FUNCTION_BLOCK FB_Kierownica
VAR_INPUT
	
			b_czujnik_wejsciowy 	:BOOL;
			b_czujnik_K1 			:BOOL;
			b_czujnik_K2 			:BOOL;
			b_czujnik_K3 			:BOOL;
			b_czujnik_K4 			:BOOL;
			b_czujnik_K5 			:BOOL;
			b_Kon2 					:BOOL;
			b_Kon1 					:BOOL;
			Zasilanie				:BOOL;
			b_Start					:BOOL;
			b_Start1				:BOOL;
			b_Stop					:BOOL;
			bS_Ready				:BOOL;
			bS_Run					:BOOL;
			bS_Done					:BOOL;
			LR_Pozycja_Zadana				:ARRAY[1..5] OF LREAL;
			b_Pobral 				:BOOL;
			int_Licznik_zadana      :INT;
			int_Kieszen_zadana 		:INT;
			automat					:BOOL;
END_VAR
VAR_OUTPUT
	
			LR_EPozycja				:LREAL;
			LR_Predkosc				:LREAL;
			bS_Enable				:BOOL;
			bS_Exe					:BOOL;
			b_Odbierz				:BOOL;
			b_Hamulec1 				:BOOL;
			b_Hamulec2 				:BOOL;
			Kier_CCW				:BOOL;
			Kier_CW					:BOOL;
END_VAR
VAR
	
			int_Kieszen				:INT :=1;
			int_Licznik				:INT; //liczenie ktora butelka w kasecie
			int_LicznikCheck		:ARRAY[1..5] OF INT; //liczenie ktora butelka w kasecie
			czas					:ARRAY[0..100] OF TON;
			Seq						:INT;
			Seq1						:INT;
			zaladowal				:BOOL;
	i: INT;
END_VAR

LR_Pozycja_Zadana[1]:=-115;	
LR_Pozycja_Zadana[2]:=-53;
LR_Pozycja_Zadana[3]:=7;
LR_Pozycja_Zadana[4]:=63;
LR_Pozycja_Zadana[5]:=122;


CASE seq OF
	

	0:
		//int_Kieszen:=1;
		
	IF (b_Start=TRUE OR b_Start1=TRUE)  AND bS_Ready=TRUE AND Zasilanie=TRUE  THEN
		b_Hamulec1:=TRUE;
		b_Hamulec2:=TRUE;
		
		IF bS_Ready=FALSE THEN 
			
			bS_Enable:=TRUE;
		END_IF
		
		
		IF bS_Ready=TRUE THEN
			seq:=5;
		END_IF
	
	
	END_IF
	
	
	5:
	
	
	
	LR_EPozycja:=LR_Pozycja_Zadana[int_Kieszen];
	LR_Predkosc:=350;
	b_Start:=FALSE;

	IF  b_Kon1=TRUE AND b_Kon2=TRUE THEN
	bS_Exe:=TRUE;
	END_IF
	
	IF bS_Run=TRUE THEN
	seq:=10;

	END_IF
	
	10:
	IF bS_Done=TRUE THEN
	bS_Exe:=FALSE;
	
	IF b_Odbierz=FALSE	THEN 
		b_Hamulec1:=FALSE;
		b_Hamulec2:=FALSE;
		
		END_IF
	seq:=0;
	
	END_IF
	


	
	
END_CASE
CASE seq1 OF
0:

			b_Start:=TRUE;
			seq1:=3;

3:
			//IF Czas[0].Q=FALSE THEN
				
			seq1:=5;
			
			//END_IF
			//int_Licznik	:=0;//zerowanie kieszeni 
			
			
5:

			IF Czas[0].Q=TRUE THEN
				
			seq1:=10;
			
			END_IF
			
10://inkremetnowanie licznika przejchala butelka 
			
			int_Licznik:=int_Licznik+1; 
			seq1:=15;
15:	
			IF int_Licznik=int_Licznik_zadana AND int_Kieszen<int_Kieszen_zadana+1 THEN
			int_Kieszen:=int_Kieszen+1;
			int_Licznik:=0;
			
			seq1:=25;	
			
			
			END_IF
		
	
			IF int_Kieszen=int_Kieszen_zadana+1 THEN
					
			GVL_GLOBAL.reset_licznik:=TRUE; ///moje
			
				b_Odbierz:=TRUE;
				int_Kieszen:=1;
				seq1:=25;	
			END_IF

			
			IF Czas[6].Q=TRUE THEN
			
						seq1:=3;
			
			END_IF
		
			

			
			
25:(*blokowanie silownika odblokowane dopiero jak przestawi sie kierownica na nastepną pozycję *)
		b_Hamulec1:=TRUE;
		b_Hamulec2:=TRUE;
		seq1:=30;	
			
30:(*startowanie serwa i czekanie jak pojedzie*)
		IF b_Kon2=TRUE AND b_Kon1=TRUE AND Czas[7].Q=TRUE THEN
			
		b_Start:=TRUE;
		seq1:=35;	
		END_IF

35:(*czekanie aż serwo wykona ruch jak wykona to skocz do 0:*)
		b_Start:=FALSE;
		
		IF bS_Done=TRUE  THEN
		seq1:=40;
		END_IF
40:(**)


		IF b_Odbierz=FALSE	THEN 
		b_Hamulec1:=FALSE;
		b_Hamulec2:=FALSE;
		seq1:=3;
		END_IF
END_CASE





Czas[0](IN:=b_czujnik_wejsciowy, PT:=T#20MS);
Czas[1](IN:=b_czujnik_K1, PT:=T#100MS);
Czas[2](IN:=b_czujnik_K2, PT:=T#100MS);
Czas[3](IN:=b_czujnik_K3, PT:=T#100MS);
Czas[4](IN:=b_czujnik_K4, PT:=T#100MS);
Czas[5](IN:=b_czujnik_K5, PT:=T#100MS);
Czas[6](IN:=b_czujnik_wejsciowy=FALSE, PT:=T#25MS);
Czas[7](IN:=seq1=30, PT:=T#500MS);
IF b_Stop=TRUE OR Zasilanie=FALSE OR automat=FALSE THEN
		
	seq:=0;
	Kier_CCW:=FALSE;
	Kier_CW:=FALSE;
	END_IF
IF b_Start1=TRUE AND Zasilanie=TRUE THEN	
	
	Kier_CCW:=TRUE;
	Kier_CW:=FALSE;
	END_IF
	IF b_pobral=TRUE THEN
		
	
	
	FOR i:=1 TO 5 BY 1 DO 
		
	int_LicznikCheck[i]:=0;
	END_FOR
 
	
	
	END_IF
	
	IF b_Pobral=TRUE THEN
			
			b_Odbierz:=FALSE;
					
			END_IF

END_FUNCTION_BLOCK

(* stored: Version 1.1.0.1, ProductVersion 3.1.4022.12
   POU FB_Kierownica: Id {79133a7a-fc9c-4f08-adb7-e5236d4321f3}, SpecialFunc None *)
